SUBAPPLICATION AX_SoftkeyOverride_TO_QXA_BG (* Digitaler AX-Ausgang mit Handbedienung: Programm-Signal (AX-Adapter OUT, ODER-verknuepft mit Softkey-Taste, solange gedrueckt) auf QXA, Background spiegelt den Zustand. Generisch. Schwester-Baustein zu MyLib::sys::SoftkeyOverride_TO_QX_BG (dort event-basiert statt AX-Adapter). *)
  (* Standard: 61499-2 *)
  (* Version 1.0, 2026-09-09, Franz Höpfinger, Meisterschulen am Ostbahnhof, Ausgelagert aus Uebung_039_sub_Outputs_AX zur Wiederverwendung. *)
  PACKAGE MyLib::sys;
  IMPORT isobus::UT::Q::const::IDs::ID_NULL;
  IMPORT logiBUS::io::DQ::logiBUS_DO;
  IMPORT logiBUS::io::DQ::logiBUS_DO_S;
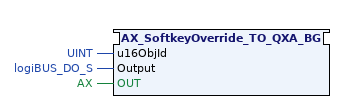
  VAR_INPUT
    u16ObjId : UINT := ID_NULL; (* Object ID Softkey/Button *)
    Output : logiBUS::io::DQ::logiBUS_DO_S := logiBUS_DO::Invalid;
  END_VAR
  SOCKETS
    OUT : adapter::types::unidirectional::AX;
  END_SOCKETS
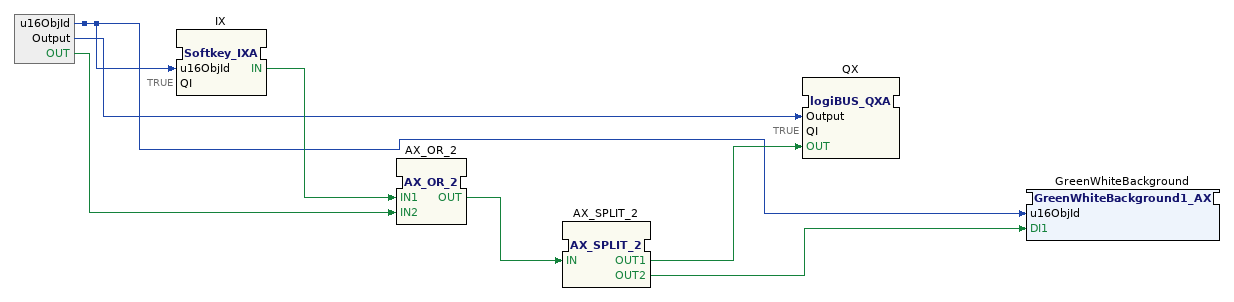
  FBS
    QX : logiBUS::io::DQ::logiBUS_QXA(QI := TRUE);
    IX : isobus::UT::io::Softkey::Softkey_IXA(QI := TRUE);
    AX_OR_2 : adapter::booleanOperators::AX_OR_2;
    AX_SPLIT_2 : adapter::events::unidirectional::AX_SPLIT_2;
  END_FBS
  SUBAPPS
    GreenWhiteBackground : MyLib::sys::GreenWhiteBackground1_AX;
  END_SUBAPPS
  DATA_CONNECTIONS
    u16ObjId TO GreenWhiteBackground.u16ObjId;
    u16ObjId TO IX.u16ObjId;
    Output TO QX.Output;
  END_CONNECTIONS
  ADAPTER_CONNECTIONS
    AX_SPLIT_2.OUT1 TO QX.OUT;
    IX.IN TO AX_OR_2.IN1;
    AX_SPLIT_2.OUT2 TO GreenWhiteBackground.DI1;
    AX_OR_2.OUT TO AX_SPLIT_2.IN;
    OUT TO AX_OR_2.IN2;
  END_CONNECTIONS
END_SUBAPPLICATION
